TYPE ST_VirtualInputs :
STRUCT
	bOnSelector : BOOL;
	bAutoSelector : BOOL;
	bStartButton : BOOL;
	bStopButton : BOOL;
	fJoystickX : LREAL;
	fJoystickY : LREAL;
END_STRUCT
END_TYPE

(* stored: Version 1.1.0.1, ProductVersion 3.1.4024.9
   DUT ST_VirtualInputs: Id {a5c51340-01ea-4684-8f4b-e6322f90d16b} *)
